TYPE udtZoneManager :
STRUCT
	Auto	:	BOOL;
	Manual	:	BOOL;
	Start	:	BOOL;
	Stop	:	BOOL;
END_STRUCT
END_TYPE

(* stored: Version 1.1.0.1, ProductVersion 3.1.4024.11
   DUT udtZoneManager: Id {a80bc0b2-d79c-4c38-99b2-dacf7a9af432} *)
